// Mitsubishi GX Works2 project: assignment2   PLC: FX3G

// global labels: Global1
VAR_GLOBAL
  Start AT X010 : BOOL;
  InventoryCheck AT M0 : BOOL;
  WorkDay AT M2 : BOOL;
  StratWorkDay AT Y010 : BOOL;
  Flour AT D1100 : INT;
  Yeast AT D1102 : INT;
  Water AT D1104 : INT;
  Oil AT D1106 : INT;
  Spices AT D1108 : INT;
END_VAR
VAR_GLOBAL CONSTANT
  FlourMin : INT := K100;
END_VAR
VAR_GLOBAL
  FlourOk : BOOL;
  YeastMin AT D1202 : INT;
  YeastOk : BOOL;
END_VAR
VAR_GLOBAL CONSTANT
  MulYeast : INT := K2;
END_VAR
VAR_GLOBAL
  MulYeastRes AT D1210 : INT;
END_VAR
VAR_GLOBAL CONSTANT
  DivYeast : INT := K10;
  MulWater : INT := K5;
END_VAR
VAR_GLOBAL
  MulWaterRes AT D1204 : INT;
END_VAR
VAR_GLOBAL CONSTANT
  DivWater : INT := K10;
END_VAR
VAR_GLOBAL
  WaterMin AT D1206 : INT;
  WaterOk : BOOL;
END_VAR
VAR_GLOBAL CONSTANT
  MulOil : INT := K3;
END_VAR
VAR_GLOBAL
  MulOilRes AT D1208 : INT;
END_VAR
VAR_GLOBAL CONSTANT
  DivOil : INT := K10;
END_VAR
VAR_GLOBAL
  OilMin AT D1213 : INT;
  OilOk : BOOL;
END_VAR
VAR_GLOBAL CONSTANT
  DivSpices : INT := K10;
END_VAR
VAR_GLOBAL
  SpicesMin AT D1215 : INT;
  SpicesOk : BOOL;
  AllOk AT M4 : BOOL;
  StartDough AT X002 : BOOL;
  DoughTimer AT TC1 : BOOL;
END_VAR
VAR_GLOBAL CONSTANT
  Sec : INT := K05;
END_VAR
VAR_GLOBAL
  DoughLight AT Y005 : BOOL;
  StartKneading AT X001 : BOOL;
  Kneading AT M14 : BOOL;
  Swelling AT M11 : BOOL;
  KeandingLight AT Y001 : BOOL;
  KneadingLight AT Y001 : BOOL;
END_VAR
VAR_GLOBAL CONSTANT
  SubFlour : INT := K100;
  SubYeast : INT := K20;
  SubWater : INT := K50;
  SubOil : INT := K30;
  SubSpices : INT := K10;
END_VAR
VAR_GLOBAL
  startswelling AT X011 : BOOL;
  SwellingTimer AT TC3 : BOOL;
  TS3 AT TS3 : BOOL;
  SwellingDone AT TS3 : BOOL;
  SwellingLight1 AT Y002 : BOOL;
  SwellingDone2 AT TS5 : BOOL;
  SwellingDone1 AT TS3 : BOOL;
  SwellingTimer1 AT TC3 : BOOL;
  SwellingTimer2 AT TC5 : BOOL;
  SwellingLight2 AT Y003 : BOOL;
END_VAR
VAR_GLOBAL CONSTANT
  CCcounter : INT := K2;
END_VAR
VAR_GLOBAL
  Bake AT M100 : BOOL;
END_VAR
VAR_GLOBAL CONSTANT
  BakeSec : INT := K40;
END_VAR
VAR_GLOBAL
  BakeLight AT Y004 : BOOL;
  CCTouch AT CC4 : BOOL;
  CsTouch AT CS4 : BOOL;
  TCSwellingTot AT TC9 : BOOL;
END_VAR
VAR_GLOBAL CONSTANT
  TotTimer : INT := K30;
END_VAR
VAR_GLOBAL
  TSSwellingTot AT TS9 : BOOL;
END_VAR
VAR_GLOBAL CONSTANT
  SecDough : INT := K30;
END_VAR
VAR_GLOBAL
  BakeTc AT TC7 : BOOL;
  BakeTs AT TS7 : BOOL;
  Control AT M22 : BOOL;
  StartQuality AT X003 : BOOL;
  analogInput2 AT D8281 : INT;
  SwellingDone4 AT D8281 : INT;
  SaveAnalog2Value AT D8000 : INT;
END_VAR
VAR_GLOBAL CONSTANT
  BiggerThen1 : INT := K200;
END_VAR
VAR_GLOBAL
  BiggerThen1Ok : BOOL;
END_VAR
VAR_GLOBAL CONSTANT
  BiggerThan1 : INT := K400;
  SmallerThan5 : INT := K2000;
END_VAR
VAR_GLOBAL
  SmallerThen5Ok : BOOL;
  BiggerThan1Ok : BOOL;
  TCSucces AT TC8 : BOOL;
END_VAR
VAR_GLOBAL CONSTANT
  TimerFive : INT := K50;
END_VAR
VAR_GLOBAL
  SuccesLight AT Y006 : BOOL;
  TSSucces AT TS8 : BOOL;
  Analog2Output AT D8282 : INT;
  CCCountTrying AT CC6 : BOOL;
END_VAR
VAR_GLOBAL CONSTANT
  CountTrying : INT := K3;
END_VAR
VAR_GLOBAL
  CsCountTrying AT CS6 : BOOL;
  Emergency AT X007 : BOOL;
  StopMachine AT M17 : BOOL;
  FlourSet AT D4444 : INT;
  YeastSet AT D4446 : INT;
  WaterSet AT D4448 : INT;
  OilSet AT D4431 : INT;
  SpicesSet AT D4433 : INT;
  M_Check AT M99 : BOOL;
  Flickering AT M20 : BOOL;
  TCFlickering AT TC20 : BOOL;
END_VAR
VAR_GLOBAL CONSTANT
  FlikeringTimer : INT := K30;
END_VAR
VAR_GLOBAL
  TSFlickering AT TS20 : BOOL;
  ControlFlikering AT M30 : BOOL;
  Flickering1 AT TC23 : BOOL;
  FlickeringTS1 AT TS23 : BOOL;
  FlickeringTC1 AT TC23 : BOOL;
  StartFlickering1 AT M70 : BOOL;
  FlickeringTC2 AT TC25 : BOOL;
  FlickeringTS2 AT TS25 : BOOL;
  StartFlickering2 AT M72 : BOOL;
  FlickeringDone AT M90 : BOOL;
  StartEmergency AT M27 : BOOL;
  StartAgain AT M55 : BOOL;
  FlourTank AT D1650 : INT;
  FlourTankRes AT D1652 : INT;
  YeastTank AT D1654 : INT;
  WaterTank AT D1656 : INT;
  OilTank AT D1658 : INT;
  SpicesTank AT D1670 : INT;
  FlourKneading AT D1672 : INT;
  YeastKneading AT D1674 : INT;
  WaterKneading AT D1676 : INT;
  OilKneading AT D1678 : INT;
  SpicesKneading AT D1680 : INT;
  Mixer AT M14 : BOOL;
  FlourSwalling AT D1682 : INT;
  FlourSwelling AT D1682 : INT;
  YeastSwelling AT D1690 : INT;
  WaterSwelling AT D1692 : INT;
  OilSwelling AT D1694 : INT;
  SpicesSwelling AT D1696 : INT;
  FlourBake AT D1698 : INT;
  YeastBake AT D1700 : INT;
  WaterBake AT D1702 : INT;
  OilBake AT D1704 : INT;
  SpicesBake AT D1706 : INT;
  BakeL AT Y004 : BOOL;
  Challah AT M112 : BOOL;
  BakeShelff AT M300 : BOOL;
END_VAR

// task Task_01 (event TRUE, interval 0, priority 31): POU_01

PROGRAM POU_01
(* structured ladder/FBD written out as ST: instructions are called as NAME(EN, inputs, outputs); _pN, _eN, _tN stand for wires *)
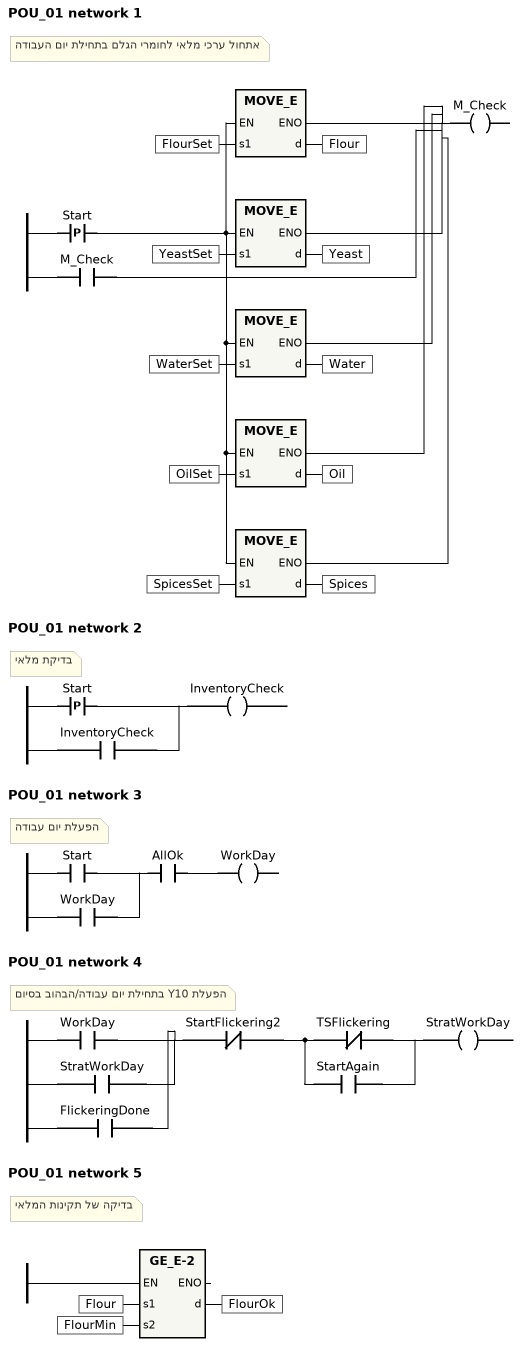
(* network 1 *)
(* אתחול ערכי מלאי לחומרי הגלם בתחילת יום העבודה *)
_p1 := LDP(TRUE, Start);
_e2 := MOVE_E(_p1, FlourSet, Flour);
_e3 := MOVE_E(_p1, YeastSet, Yeast);
_e4 := MOVE_E(_p1, WaterSet, Water);
_e5 := MOVE_E(_p1, OilSet, Oil);
_e6 := MOVE_E(_p1, SpicesSet, Spices);
M_Check := _e2 OR _e3 OR _e4 OR _e5 OR _e6 OR M_Check;
(* network 2 *)
(* בדיקת מלאי *)
InventoryCheck := LDP(TRUE, Start) OR InventoryCheck;
(* network 3 *)
(* הפעלת יום עבודה *)
WorkDay := (Start OR WorkDay) AND AllOk;
(* network 4 *)
(* הפעלת Y10 בתחילת יום עבודה/הבהוב בסיום *)
_p1 := (WorkDay OR StratWorkDay OR FlickeringDone) AND NOT StartFlickering2;
StratWorkDay := (_p1 AND NOT TSFlickering) OR (_p1 AND StartAgain);
(* network 5 *)
(* בדיקה של תקינות המלאי *)
GE_E(TRUE, Flour, FlourMin, FlourOk);
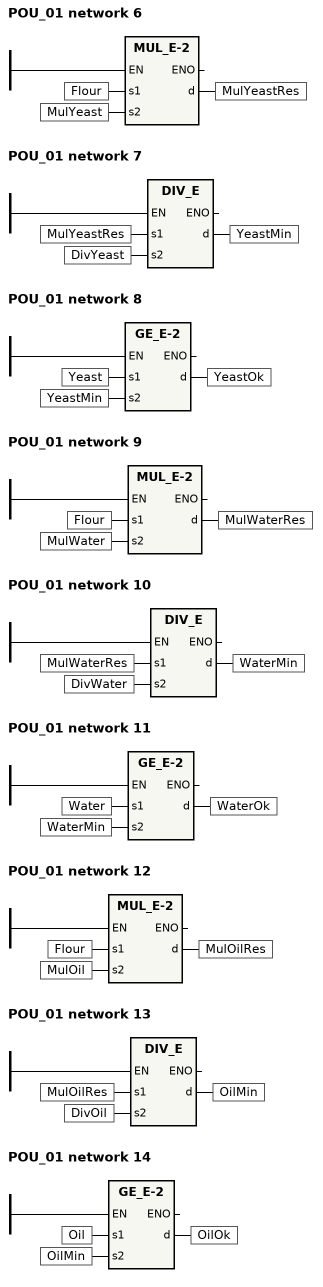
(* network 6 *)
MUL_E(TRUE, Flour, MulYeast, MulYeastRes);
(* network 7 *)
DIV_E(TRUE, MulYeastRes, DivYeast, YeastMin);
(* network 8 *)
GE_E(TRUE, Yeast, YeastMin, YeastOk);
(* network 9 *)
MUL_E(TRUE, Flour, MulWater, MulWaterRes);
(* network 10 *)
DIV_E(TRUE, MulWaterRes, DivWater, WaterMin);
(* network 11 *)
GE_E(TRUE, Water, WaterMin, WaterOk);
(* network 12 *)
MUL_E(TRUE, Flour, MulOil, MulOilRes);
(* network 13 *)
DIV_E(TRUE, MulOilRes, DivOil, OilMin);
(* network 14 *)
GE_E(TRUE, Oil, OilMin, OilOk);
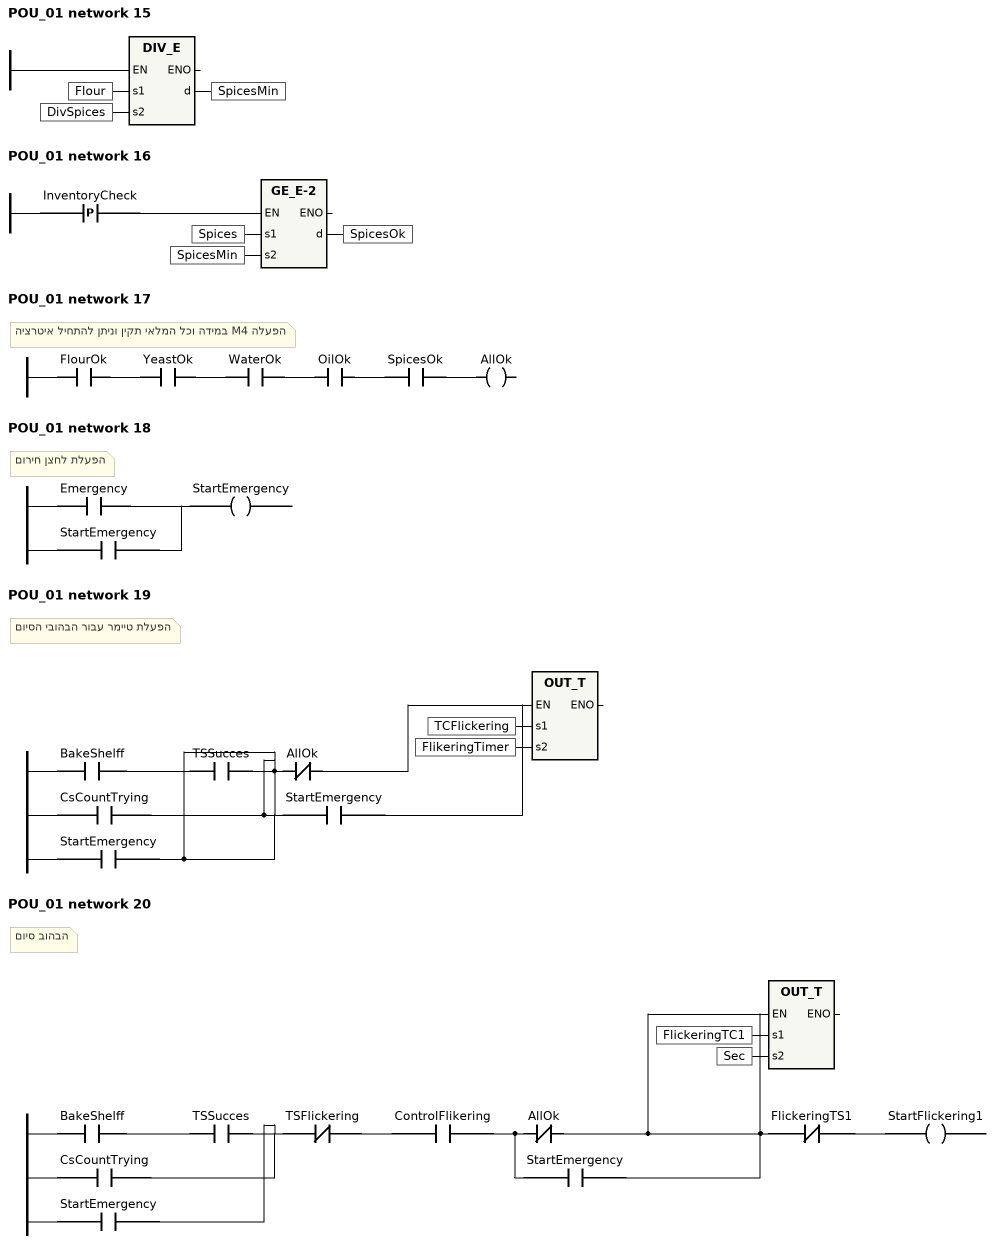
(* network 15 *)
DIV_E(TRUE, Flour, DivSpices, SpicesMin);
(* network 16 *)
GE_E(LDP(TRUE, InventoryCheck), Spices, SpicesMin, SpicesOk);
(* network 17 *)
(* הפעלה M4 במידה וכל המלאי תקין וניתן להתחיל איטרציה *)
AllOk := FlourOk AND YeastOk AND WaterOk AND OilOk AND SpicesOk;
(* network 18 *)
(* הפעלת לחצן חירום *)
StartEmergency := Emergency OR StartEmergency;
(* network 19 *)
(* הפעלת טיימר עבור הבהובי הסיום *)
_p1 := (BakeShelff AND TSSucces) OR CsCountTrying OR StartEmergency;
OUT_T((_p1 AND NOT AllOk) OR (_p1 AND StartEmergency), TCFlickering, FlikeringTimer);
(* network 20 *)
(* הבהוב סיום *)
_p1 := (((BakeShelff AND TSSucces) OR CsCountTrying OR StartEmergency) AND NOT TSFlickering) AND ControlFlikering;
_p2 := (_p1 AND NOT AllOk) OR (_p1 AND StartEmergency);
OUT_T(_p2, FlickeringTC1, Sec);
StartFlickering1 := _p2 AND NOT FlickeringTS1;
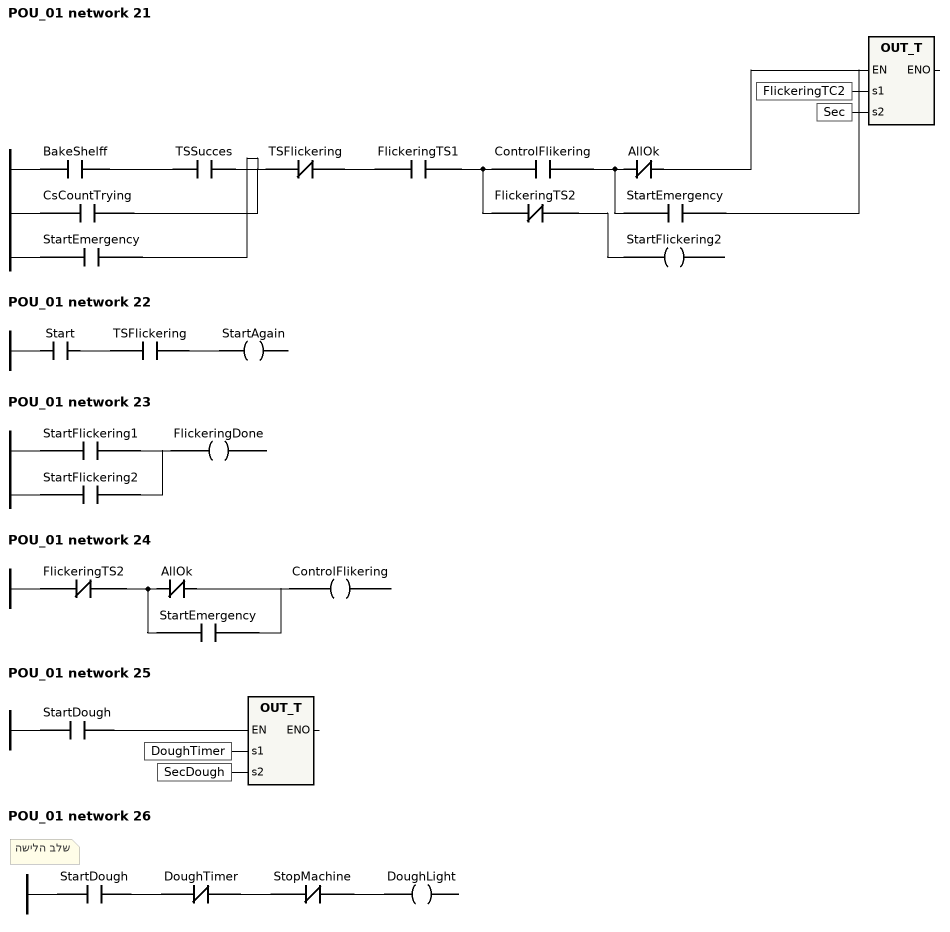
(* network 21 *)
_p1 := (((BakeShelff AND TSSucces) OR CsCountTrying OR StartEmergency) AND NOT TSFlickering) AND FlickeringTS1;
_p2 := _p1 AND ControlFlikering;
OUT_T((_p2 AND NOT AllOk) OR (_p2 AND StartEmergency), FlickeringTC2, Sec);
StartFlickering2 := _p1 AND NOT FlickeringTS2;
(* network 22 *)
StartAgain := Start AND TSFlickering;
(* network 23 *)
FlickeringDone := StartFlickering1 OR StartFlickering2;
(* network 24 *)
_p1 := NOT FlickeringTS2;
ControlFlikering := (_p1 AND NOT AllOk) OR (_p1 AND StartEmergency);
(* network 25 *)
OUT_T(StartDough, DoughTimer, SecDough);
(* network 26 *)
(* שלב הלישה *)
DoughLight := StartDough AND NOT DoughTimer AND NOT StopMachine;
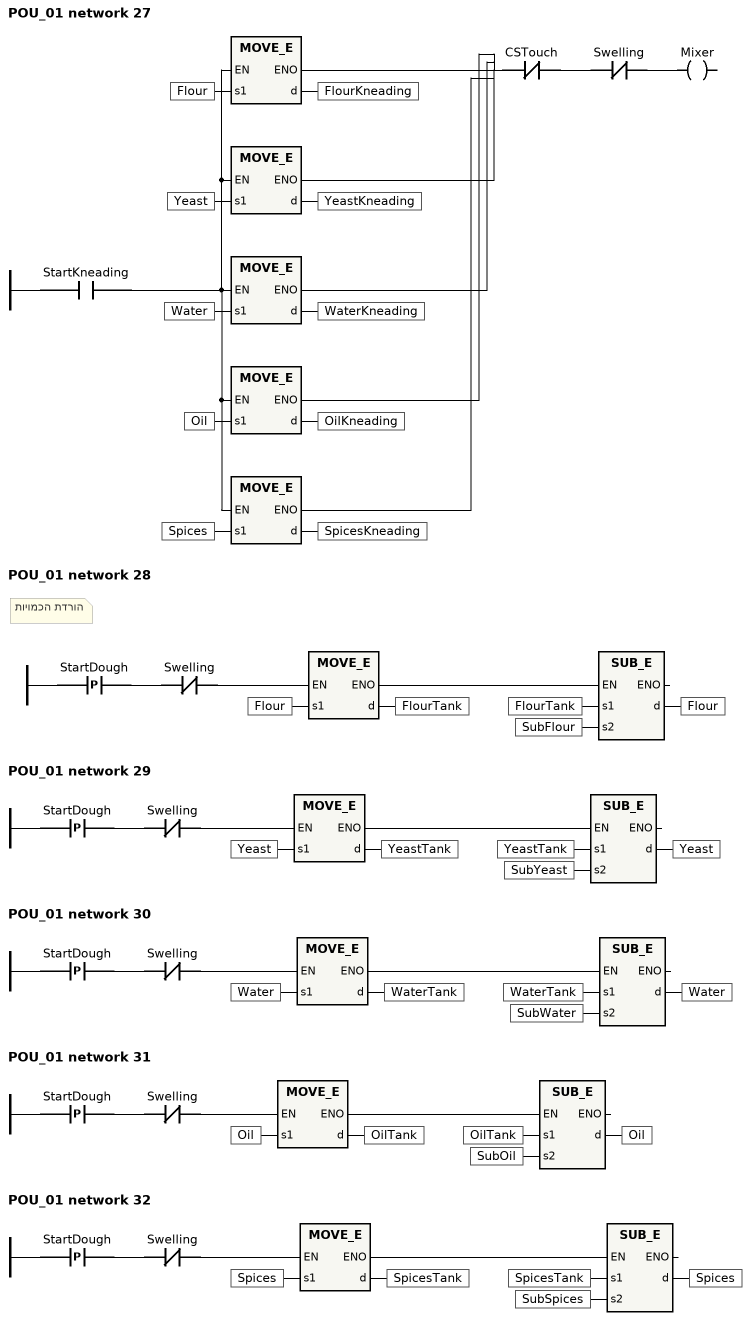
(* network 27 *)
_e1 := MOVE_E(StartKneading, Flour, FlourKneading);
_e2 := MOVE_E(StartKneading, Yeast, YeastKneading);
_e3 := MOVE_E(StartKneading, Water, WaterKneading);
_e4 := MOVE_E(StartKneading, Oil, OilKneading);
_e5 := MOVE_E(StartKneading, Spices, SpicesKneading);
Mixer := ((_e1 OR _e2 OR _e3 OR _e4 OR _e5) AND NOT CSTouch) AND NOT Swelling;
(* network 28 *)
(* הורדת הכמויות *)
_e1 := MOVE_E(LDP(TRUE, StartDough) AND NOT Swelling, Flour, FlourTank);
SUB_E(_e1, FlourTank, SubFlour, Flour);
(* network 29 *)
_e1 := MOVE_E(LDP(TRUE, StartDough) AND NOT Swelling, Yeast, YeastTank);
SUB_E(_e1, YeastTank, SubYeast, Yeast);
(* network 30 *)
_e1 := MOVE_E(LDP(TRUE, StartDough) AND NOT Swelling, Water, WaterTank);
SUB_E(_e1, WaterTank, SubWater, Water);
(* network 31 *)
_e1 := MOVE_E(LDP(TRUE, StartDough) AND NOT Swelling, Oil, OilTank);
SUB_E(_e1, OilTank, SubOil, Oil);
(* network 32 *)
_e1 := MOVE_E(LDP(TRUE, StartDough) AND NOT Swelling, Spices, SpicesTank);
SUB_E(_e1, SpicesTank, SubSpices, Spices);
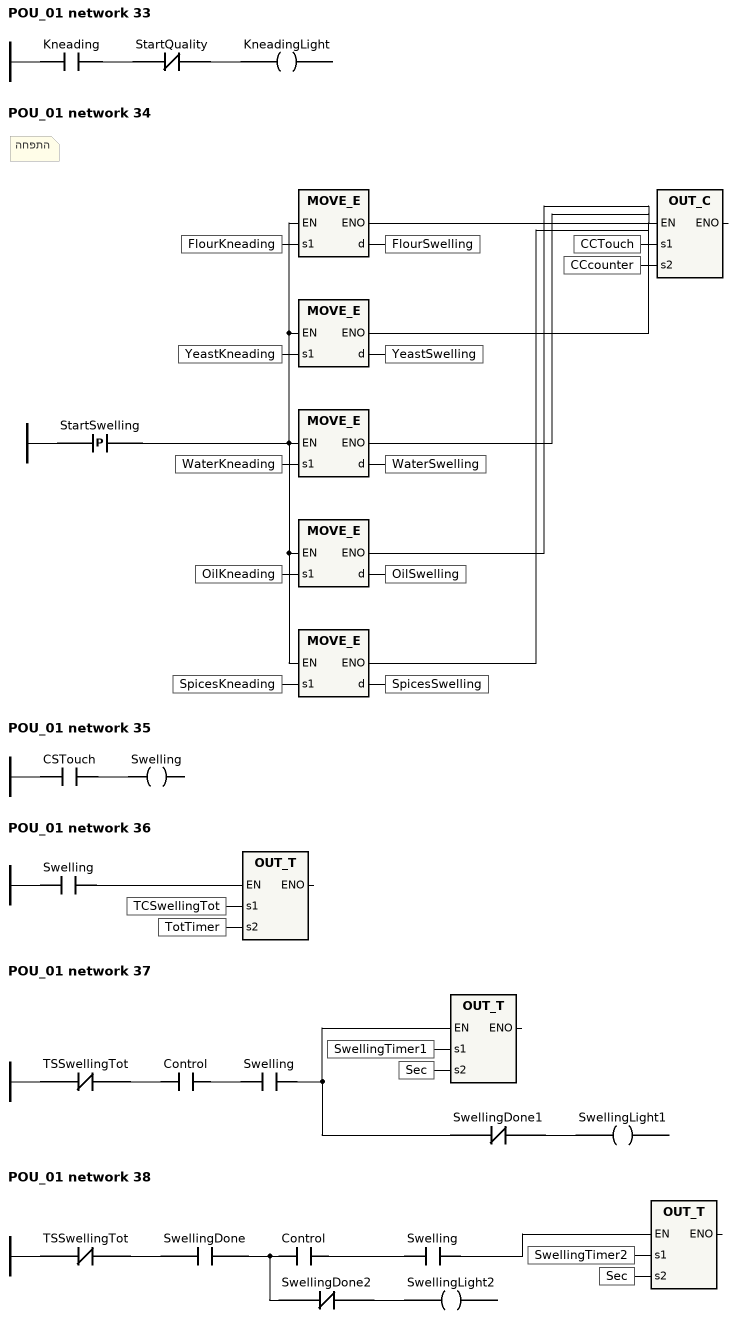
(* network 33 *)
KneadingLight := Kneading AND NOT StartQuality;
(* network 34 *)
(* התפחה *)
_p1 := LDP(TRUE, StartSwelling);
_e2 := MOVE_E(_p1, FlourKneading, FlourSwelling);
_e3 := MOVE_E(_p1, YeastKneading, YeastSwelling);
_e4 := MOVE_E(_p1, WaterKneading, WaterSwelling);
_e5 := MOVE_E(_p1, OilKneading, OilSwelling);
_e6 := MOVE_E(_p1, SpicesKneading, SpicesSwelling);
OUT_C(_e2 OR _e3 OR _e4 OR _e5 OR _e6, CCTouch, CCcounter);
(* network 35 *)
Swelling := CSTouch;
(* network 36 *)
OUT_T(Swelling, TCSwellingTot, TotTimer);
(* network 37 *)
_p1 := NOT TSSwellingTot AND Control AND Swelling;
OUT_T(_p1, SwellingTimer1, Sec);
SwellingLight1 := _p1 AND NOT SwellingDone1;
(* network 38 *)
_p1 := NOT TSSwellingTot AND SwellingDone;
OUT_T(_p1 AND Control AND Swelling, SwellingTimer2, Sec);
SwellingLight2 := _p1 AND NOT SwellingDone2;
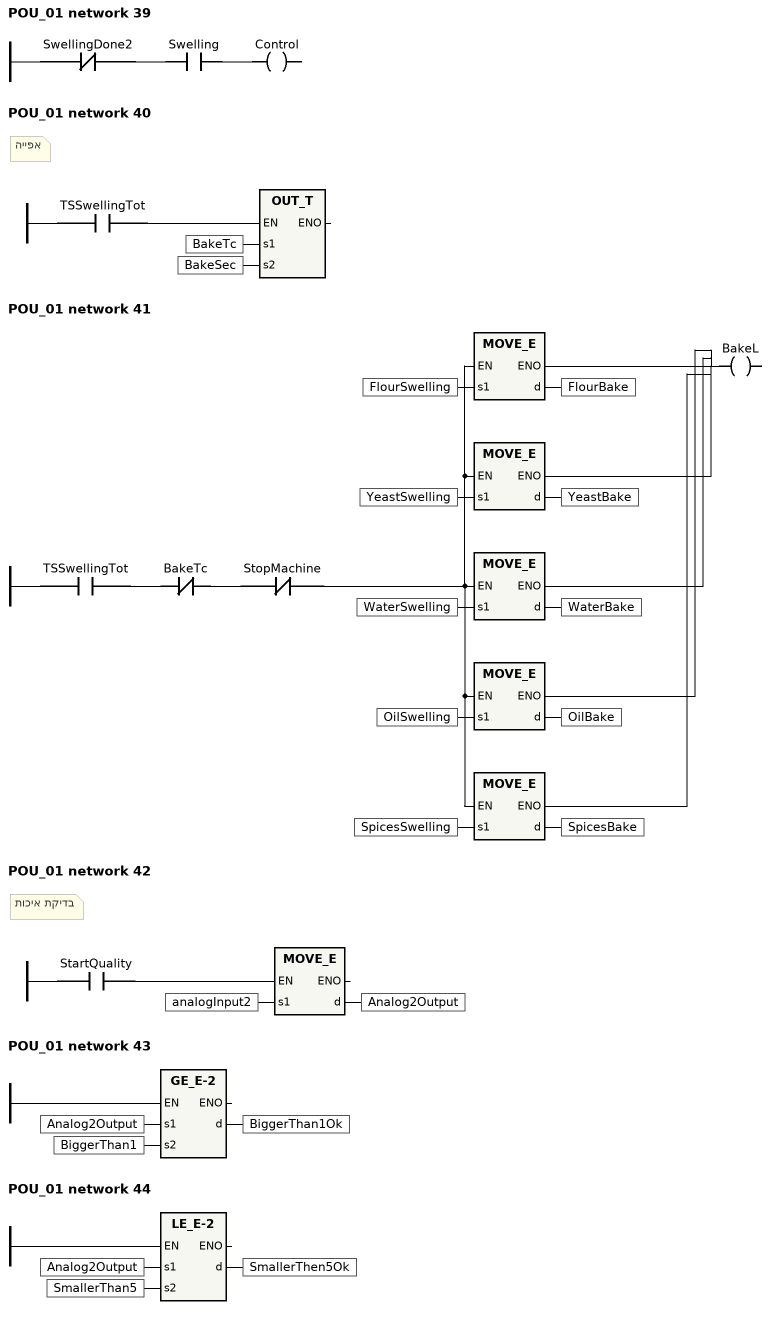
(* network 39 *)
Control := NOT SwellingDone2 AND Swelling;
(* network 40 *)
(* אפייה *)
OUT_T(TSSwellingTot, BakeTc, BakeSec);
(* network 41 *)
_p1 := TSSwellingTot AND NOT BakeTc AND NOT StopMachine;
_e2 := MOVE_E(_p1, FlourSwelling, FlourBake);
_e3 := MOVE_E(_p1, YeastSwelling, YeastBake);
_e4 := MOVE_E(_p1, WaterSwelling, WaterBake);
_e5 := MOVE_E(_p1, OilSwelling, OilBake);
_e6 := MOVE_E(_p1, SpicesSwelling, SpicesBake);
BakeL := _e2 OR _e3 OR _e4 OR _e5 OR _e6;
(* network 42 *)
(* בדיקת איכות *)
MOVE_E(StartQuality, analogInput2, Analog2Output);
(* network 43 *)
GE_E(TRUE, Analog2Output, BiggerThan1, BiggerThan1Ok);
(* network 44 *)
LE_E(TRUE, Analog2Output, SmallerThan5, SmallerThen5Ok);
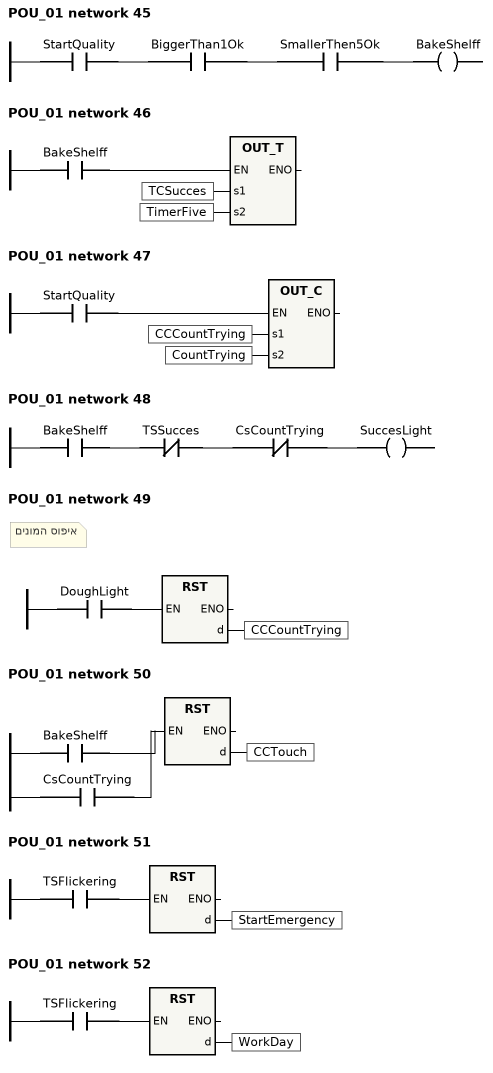
(* network 45 *)
BakeShelff := StartQuality AND BiggerThan1Ok AND SmallerThen5Ok;
(* network 46 *)
OUT_T(BakeShelff, TCSucces, TimerFive);
(* network 47 *)
OUT_C(StartQuality, CCCountTrying, CountTrying);
(* network 48 *)
SuccesLight := BakeShelff AND NOT TSSucces AND NOT CsCountTrying;
(* network 49 *)
(* איפוס המונים *)
RST(DoughLight, CCCountTrying);
(* network 50 *)
RST(BakeShelff OR CsCountTrying, CCTouch);
(* network 51 *)
RST(TSFlickering, StartEmergency);
(* network 52 *)
RST(TSFlickering, WorkDay);
END_PROGRAM
